KUKA KRL program: tool01_chk.src, tool01_chk.dat

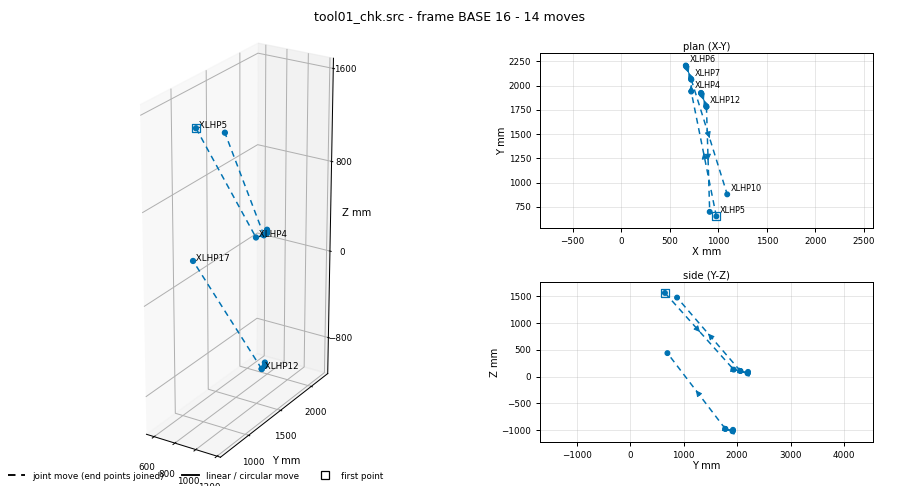
[picture p0: tool path of tool01_chk.src in frame BASE 16, 14 of 17 moves have a stored position in this frame; points joined in program order, loops and branches not executed]
--- tool01_chk.src ---
&ACCESS RVP
&REL 64
&COMMENT Werkzeugpruefprogramm
&PARAM TEMPLATE = C:\KRC\ROBOTER\TEMPLATE\VG_HP
&PARAM EDITMASK = *
DEF TOOL01_chk( )
;FOLD INI
;FOLD BASISTECH INI
    GLOBAL INTERRUPT DECL 3 WHEN $STOPMESS==TRUE DO IR_STOPM ( )
    INTERRUPT ON 3
    BAS (#INITMOV,0 )
;ENDFOLD (BASISTECH INI)
;FOLD SPOTTECH INI
    USERSPOT(#INIT)
;ENDFOLD (SPOTTECH INI)
;FOLD GRIPPERTECH INI
    USER_GRP(0,DUMMY,DUMMY,GDEFAULT)
;ENDFOLD (GRIPPERTECH INI)
;FOLD USER INI
;Make your modifications here
;FOLD COLLISION_V_3.01 INI ;%{E}
    IF (COLLISION_DATA[1].I_NR>0) THEN
    GLOBAL INTERRUPT DECL 21 WHEN $IN[COLLISION_DATA[1].I_NR]==FALSE DO COLLSTOP (1,0 )
    ENDIF
    IF (COLLISION_DATA[2].I_NR>0) THEN
    GLOBAL INTERRUPT DECL 22 WHEN $IN[COLLISION_DATA[2].I_NR]==FALSE DO COLLSTOP (2,0 )
    ENDIF
    IF (COLLISION_DATA[3].I_NR>0) THEN
    GLOBAL INTERRUPT DECL 23 WHEN $IN[COLLISION_DATA[3].I_NR]==FALSE DO COLLSTOP (3,0 )
    ENDIF
    IF (COLLISION_DATA[4].I_NR>0) THEN
    GLOBAL INTERRUPT DECL 24 WHEN $IN[COLLISION_DATA[4].I_NR]==FALSE DO COLLSTOP (4,0 )
    ENDIF
;ENDFOLD (Collision)
;ENDFOLD (USER INI)
;ENDFOLD (INI)
;FOLD ; Anlagenbezeichn:               Stations-Nr:;%{PE}%R 5.2.7,%MKUKATPBASIS,%CCOMMENT,%VNORMAL,%P 2:Anlagenbezeichn:               Stations-Nr:
;ENDFOLD
;FOLD ; Stand / Version:;%{PE}%R 5.2.7,%MKUKATPBASIS,%CCOMMENT,%VNORMAL,%P 2:Stand / Version:
;ENDFOLD
;FOLD ; Name Bearbeiter:;%{PE}%R 5.2.7,%MKUKATPBASIS,%CCOMMENT,%VNORMAL,%P 2:Name Bearbeiter:
;ENDFOLD
;Sicherheitsfrage (nur im Musterprogramm, nach teachen entfernen)
wait for false
;FOLD ; ***************************************;%{PE}%R 2.4.6,%MKUKATPBASIS,%CCOMMENT,%VNORMAL,%P 2:***************************************
;ENDFOLD
;FOLD ; A C H T U N G  ! ! !   Nur in T1 fahren;%{PE}%R 2.4.6,%MKUKATPBASIS,%CCOMMENT,%VNORMAL,%P 2:A C H T U N G  ! ! !   Nur in T1 fahren
;ENDFOLD
;FOLD ; ***************************************;%{PE}%R 2.4.6,%MKUKATPBASIS,%CCOMMENT,%VNORMAL,%P 2:***************************************
;ENDFOLD
WAIT FOR $T1
;Wenn notwendig vorher das Werkzeug im Bahnhof ablegen
;Roboterpruefprogramm
rob_ok ( )
;Wenn notwendig zu pruefendes Werkzeug ankoppeln
;FOLD PTP HOME  Vel= 100 % DEFAULT;%{PE}%R 3.2.43,%MKUKATPBASIS,%CMOVE,%VPTP,%P 1:PTP, 2:HOME, 3:, 5:100, 7:DEFAULT
$BWDSTART = FALSE
PDAT_ACT=PDEFAULT
BAS(#PTP_DAT)
FDAT_ACT=FHOME
BAS(#FRAMES)
BAS(#VEL_PTP,100)
$H_POS=XHOME
PTP XHOME
;ENDFOLD
;FOLD PTP LHP5  Vel= 100 % PDAT Tool[16] Base[16];%{PE}%R 3.2.43,%MKUKATPBASIS,%CMOVE,%VPTP,%P 1:PTP, 2:LHP5, 3:, 5:100, 7:PDAT
    $BWDSTART = FALSE
    PDAT_ACT=PPDAT
    BAS(#PTP_DAT)
    FDAT_ACT=FLHP5
    BAS(#FRAMES)
    BAS(#VEL_PTP,100)
    PTP XLHP5
;ENDFOLD
;FOLD PTP LHP4  Vel= 100 % PDAT Tool[16] Base[16];%{PE}%R 3.2.43,%MKUKATPBASIS,%CMOVE,%VPTP,%P 1:PTP, 2:LHP4, 3:, 5:100, 7:PDAT
    $BWDSTART = FALSE
    PDAT_ACT=PPDAT
    BAS(#PTP_DAT)
    FDAT_ACT=FLHP4
    BAS(#FRAMES)
    BAS(#VEL_PTP,100)
    PTP XLHP4
;ENDFOLD
;FOLD PTP LHP7  Vel= 100 % PDAT Tool[16] Base[16];%{PE}%R 3.2.43,%MKUKATPBASIS,%CMOVE,%VPTP,%P 1:PTP, 2:LHP7, 3:, 5:100, 7:PDAT
    $BWDSTART = FALSE
    PDAT_ACT=PPDAT
    BAS(#PTP_DAT)
    FDAT_ACT=FLHP7
    BAS(#FRAMES)
    BAS(#VEL_PTP,100)
    PTP XLHP7
;ENDFOLD
;FOLD PTP LHP6  Vel= 100 % PDAT Tool[16] Base[16];%{PE}%R 3.2.43,%MKUKATPBASIS,%CMOVE,%VPTP,%P 1:PTP, 2:LHP6, 3:, 5:100, 7:PDAT
    $BWDSTART = FALSE
    PDAT_ACT=PPDAT
    BAS(#PTP_DAT)
    FDAT_ACT=FLHP6
    BAS(#FRAMES)
    BAS(#VEL_PTP,100)
    PTP XLHP6
;ENDFOLD
;FOLD ; 1.Kontrollposition mit Tool 16;%{PE}%R 5.2.17,%MKUKATPBASIS,%CCOMMENT,%VNORMAL,%P 2:1.Kontrollposition mit Tool 16
;ENDFOLD
;FOLD ; Pruefspitze - Werkzeugspitze bzw. Greiferreferenzpunkt;%{PE}%R 2.4.6,%MKUKATPBASIS,%CCOMMENT,%VNORMAL,%P 2:Pruefspitze - Werkzeugspitze bzw. Greiferreferenzpunkt
;ENDFOLD
;FOLD ; Spitze unten;%{PE}%R 2.4.6,%MKUKATPBASIS,%CCOMMENT,%VNORMAL,%P 2:Spitze unten
;ENDFOLD
;FOLD LIN Kontroll1  Vel= 1 m/s CPDAT Tool[16] Base[16];%{PE}%R 3.2.43,%MKUKATPBASIS,%CMOVE,%VLIN,%P 1:LIN, 2:Kontroll1, 3:, 5:1, 7:CPDAT
    $BWDSTART = FALSE
    LDAT_ACT=LCPDAT
    BAS(#CP_DAT)
    FDAT_ACT=FKontroll1
    BAS(#FRAMES)
    BAS(#VEL_CP,1)
    LIN XKontroll1
;ENDFOLD
WAIT FOR  $IN[1026]==TRUE ; Kontrollposition Werkzeug mit Tool16 (Nullwerkzeug)
;PTP LHP freifahren
;FOLD LIN LHP8  Vel= 2 m/s CPDAT Tool[16] Base[16];%{PE}%R 3.2.43,%MKUKATPBASIS,%CMOVE,%VLIN,%P 1:LIN, 2:LHP8, 3:, 5:2, 7:CPDAT
    $BWDSTART = FALSE
    LDAT_ACT=LCPDAT
    BAS(#CP_DAT)
    FDAT_ACT=FLHP8
    BAS(#FRAMES)
    BAS(#VEL_CP,2)
    LIN XLHP8
;ENDFOLD
;FOLD PTP LHP9  Vel= 100 % PDAT Tool[16] Base[16];%{PE}%R 3.2.43,%MKUKATPBASIS,%CMOVE,%VPTP,%P 1:PTP, 2:LHP9, 3:, 5:100, 7:PDAT
    $BWDSTART = FALSE
    PDAT_ACT=PPDAT
    BAS(#PTP_DAT)
    FDAT_ACT=FLHP9
    BAS(#FRAMES)
    BAS(#VEL_PTP,100)
    PTP XLHP9
;ENDFOLD
;FOLD PTP LHP10  Vel= 100 % PDAT Tool[16] Base[16];%{PE}%R 3.2.43,%MKUKATPBASIS,%CMOVE,%VPTP,%P 1:PTP, 2:LHP10, 3:, 5:100, 7:PDAT
    $BWDSTART = FALSE
    PDAT_ACT=PPDAT
    BAS(#PTP_DAT)
    FDAT_ACT=FLHP10
    BAS(#FRAMES)
    BAS(#VEL_PTP,100)
    PTP XLHP10
;ENDFOLD
;Wichtig: auf Home zurueck fahren und auf aktuelles TOOL umschalten
;FOLD PTP HOME  Vel= 100 % PDAT;%{PE}%R 3.2.43,%MKUKATPBASIS,%CMOVE,%VPTP,%P 1:PTP, 2:HOME, 3:, 5:100, 7:PDAT
    $BWDSTART = FALSE
    PDAT_ACT=PPDAT
    BAS(#PTP_DAT)
    FDAT_ACT=FHOME
    BAS(#FRAMES)
    BAS(#VEL_PTP,100)
    $H_POS=XHOME
    PTP XHOME
;ENDFOLD
;FOLD PTP LHP12  Vel= 100 % PDAT Tool[1] Base[16];%{PE}%R 3.2.43,%MKUKATPBASIS,%CMOVE,%VPTP,%P 1:PTP, 2:LHP12, 3:, 5:100, 7:PDAT
    $BWDSTART = FALSE
    PDAT_ACT=PPDAT
    BAS(#PTP_DAT)
    FDAT_ACT=FLHP12
    BAS(#FRAMES)
    BAS(#VEL_PTP,100)
    PTP XLHP12
;ENDFOLD
;FOLD PTP LHP13  Vel= 100 % PDAT Tool[1] Base[16];%{PE}%R 3.2.43,%MKUKATPBASIS,%CMOVE,%VPTP,%P 1:PTP, 2:LHP13, 3:, 5:100, 7:PDAT
    $BWDSTART = FALSE
    PDAT_ACT=PPDAT
    BAS(#PTP_DAT)
    FDAT_ACT=FLHP13
    BAS(#FRAMES)
    BAS(#VEL_PTP,100)
    PTP XLHP13
;ENDFOLD
;FOLD ; 2.Kontrollposition mit Tool aktuell;%{PE}%R 5.2.17,%MKUKATPBASIS,%CCOMMENT,%VNORMAL,%P 2:2.Kontrollposition mit Tool aktuell
;ENDFOLD
;FOLD ; Pruefspitze - Werkzeugspitze bzw. Greiferreferenzpunkt;%{PE}%R 2.4.6,%MKUKATPBASIS,%CCOMMENT,%VNORMAL,%P 2:Pruefspitze - Werkzeugspitze bzw. Greiferreferenzpunkt
;ENDFOLD
;FOLD ; Spitze unten;%{PE}%R 2.4.6,%MKUKATPBASIS,%CCOMMENT,%VNORMAL,%P 2:Spitze unten
;ENDFOLD
;PTP KONTROLL2 teachen mit dem zugehoerigen Tool
;FOLD LIN Kontroll2  Vel= 1 m/s CPDAT Tool[1] Base[16];%{PE}%R 3.2.43,%MKUKATPBASIS,%CMOVE,%VLIN,%P 1:LIN, 2:Kontroll2, 3:, 5:1, 7:CPDAT
    $BWDSTART = FALSE
    LDAT_ACT=LCPDAT
    BAS(#CP_DAT)
    FDAT_ACT=FKontroll2
    BAS(#FRAMES)
    BAS(#VEL_CP,1)
    LIN XKontroll2
;ENDFOLD
WAIT FOR  $IN[1026]==TRUE ; Kontrollposition Werkzeug mit zugehoerigem Tool
;PTP LHP zur Ausgangsstellung
;FOLD LIN LHP15  Vel= 1 m/s CPDAT Tool[1] Base[16];%{PE}%R 3.2.43,%MKUKATPBASIS,%CMOVE,%VLIN,%P 1:LIN, 2:LHP15, 3:, 5:1, 7:CPDAT
    $BWDSTART = FALSE
    LDAT_ACT=LCPDAT
    BAS(#CP_DAT)
    FDAT_ACT=FLHP15
    BAS(#FRAMES)
    BAS(#VEL_CP,1)
    LIN XLHP15
;ENDFOLD
;FOLD PTP LHP16  Vel= 100 % PDAT Tool[1] Base[16];%{PE}%R 3.2.43,%MKUKATPBASIS,%CMOVE,%VPTP,%P 1:PTP, 2:LHP16, 3:, 5:100, 7:PDAT
    $BWDSTART = FALSE
    PDAT_ACT=PPDAT
    BAS(#PTP_DAT)
    FDAT_ACT=FLHP16
    BAS(#FRAMES)
    BAS(#VEL_PTP,100)
    PTP XLHP16
;ENDFOLD
;FOLD PTP LHP17  Vel= 100 % PDAT Tool[1] Base[16];%{PE}%R 3.2.43,%MKUKATPBASIS,%CMOVE,%VPTP,%P 1:PTP, 2:LHP17, 3:, 5:100, 7:PDAT
    $BWDSTART = FALSE
    PDAT_ACT=PPDAT
    BAS(#PTP_DAT)
    FDAT_ACT=FLHP17
    BAS(#FRAMES)
    BAS(#VEL_PTP,100)
    PTP XLHP17
;ENDFOLD
;FOLD PTP HOME  Vel= 100 % DEFAULT;%{PE}%R 3.2.43,%MKUKATPBASIS,%CMOVE,%VPTP,%P 1:PTP, 2:HOME, 3:, 5:100, 7:DEFAULT
    $BWDSTART = FALSE
    PDAT_ACT=PDEFAULT
    BAS(#PTP_DAT)
    FDAT_ACT=FHOME
    BAS(#FRAMES)
    BAS(#VEL_PTP,100)
    $H_POS=XHOME
    PTP XHOME
;ENDFOLD
;Wenn notwendig das ursprüngliche Werkzeug wieder ankoppeln
END

--- tool01_chk.dat ---
&ACCESS RVP
&REL 64
&COMMENT Werkzeugpruefprogramm
&PARAM TEMPLATE = C:\KRC\ROBOTER\TEMPLATE\VG_HP
&PARAM EDITMASK = *
DEFDAT  TOOL01_CHK
;FOLD EXTERNAL DECLARATIONS;%{PE}%V3.2.0,%MKUKATPBASIS,%CEXT,%VCOMMON,%P
;ENDFOLD

DECL BASIS_SUGG_T LAST_BASIS={POINT1[] "P0                      ",POINT2[] "P0                      ",CP_PARAMS[] "CPDAT0                  ",PTP_PARAMS[] "PDAT0                  ",CONT[] "                        ",CP_VEL[] "2                       ",PTP_VEL[] "100                     "}
DECL E6POS XLHP1={x 980.162,y 652.3817,z 1564.854,a 159.7475,b -4.016941,c 179.1242,s 18,t 43,e1 -100.6665,e2 0.0,e3 0.0,e4 0.0,e5 0.0,e6 0.0}
DECL E6POS XKONTROLL1={x 665.4379,y 2205.945,z 89.04919,a -69.02276,b -16.31656,c -177.4203,s 18,t 3,e1 -100.6661,e2 0.0,e3 0.0,e4 0.0,e5 0.0,e6 0.0}
DECL E6POS XLHP4={x 721.3241,y 1937.913,z 131.173,a -69.07279,b -16.22725,c -174.2469,s 18,t 3,e1 -100.6665,e2 0.0,e3 0.0,e4 0.0,e5 0.0,e6 0.0}
DECL E6POS XLHP5={x 980.1787,y 652.3956,z 1564.878,a 159.749,b -4.016594,c 179.1235,s 18,t 43,e1 -100.6665,e2 0.0,e3 0.0,e4 0.0,e5 0.0,e6 0.0}
DECL E6POS XKONTROLL2={x 821.7288,y 1924.512,z -993.7808,a 111.0075,b 16.30128,c -2.863059,s 18,t 3,e1 -100.6665,e2 0.0,e3 0.0,e4 0.0,e5 0.0,e6 0.0}
DECL E6POS XLHP6={x 669.3153,y 2199.305,z 63.11586,a -69.03085,b -16.31788,c -177.4184,s 18,t 3,e1 -100.6665,e2 0.0,e3 0.0,e4 0.0,e5 0.0,e6 0.0}
DECL E6POS XLHP7={x 721.9332,y 2061.901,z 106.2138,a -69.02566,b -16.3192,c -177.4167,s 18,t 3,e1 -100.6665,e2 0.0,e3 0.0,e4 0.0,e5 0.0,e6 0.0}
DECL E6POS XLHP8={x 669.3173,y 2199.294,z 63.11121,a -69.03092,b -16.31823,c -177.4184,s 18,t 3,e1 -100.6665,e2 0.0,e3 0.0,e4 0.0,e5 0.0,e6 0.0}
DECL E6POS XLHP9={x 721.9332,y 2061.901,z 106.2138,a -69.02566,b -16.3192,c -177.4167,s 18,t 3,e1 -100.6665,e2 0.0,e3 0.0,e4 0.0,e5 0.0,e6 0.0}
DECL E6POS XLHP10={x 1092.313,y 878.8538,z 1478.174,a 177.4667,b -3.04429,c -178.5137,s 18,t 43,e1 -100.6665,e2 0.0,e3 0.0,e4 0.0,e5 0.0,e6 0.0}
DECL E6POS XLHP12={x 878.2603,y 1780.715,z -976.2581,a 111.0027,b 16.29478,c -2.869996,s 18,t 3,e1 -100.6665,e2 0.0,e3 0.0,e4 0.0,e5 0.0,e6 0.0}
DECL E6POS XLHP13={x 825.5921,y 1917.879,z -1019.667,a 111.0074,b 16.30032,c -2.863573,s 18,t 3,e1 -100.6665,e2 0.0,e3 0.0,e4 0.0,e5 0.0,e6 0.0}
DECL E6POS XLHP15={x 825.5995,y 1917.881,z -1019.669,a 111.007,b 16.29994,c -2.863638,s 18,t 3,e1 -100.6665,e2 0.0,e3 0.0,e4 0.0,e5 0.0,e6 0.0}
DECL E6POS XLHP16={x 878.2797,y 1780.88,z -976.2927,a 111.0091,b 16.29242,c -2.869744,s 18,t 3,e1 -100.6665,e2 0.0,e3 0.0,e4 0.0,e5 0.0,e6 0.0}
DECL E6POS XLHP17={x 911.847,y 698.7325,z 439.7753,a -20.25009,b 3.988059,c 0.4698318,s 18,t 43,e1 -100.6665,e2 0.0,e3 0.0,e4 0.0,e5 0.0,e6 0.0}
DECL FDAT FLHP1={TOOL_NO 16,BASE_NO 16,IPO_FRAME #BASE}
DECL FDAT FKONTROLL1={TOOL_NO 16,BASE_NO 16,IPO_FRAME #BASE}
DECL FDAT FLHP4={TOOL_NO 16,BASE_NO 16,IPO_FRAME #BASE}
DECL FDAT FLHP5={TOOL_NO 16,BASE_NO 16,IPO_FRAME #BASE}
DECL FDAT FKontroll2={TOOL_NO 1,BASE_NO 16,IPO_FRAME #BASE}
DECL FDAT FLHP6={TOOL_NO 16,BASE_NO 16,IPO_FRAME #BASE}
DECL FDAT FLHP7={TOOL_NO 16,BASE_NO 16,IPO_FRAME #BASE}
DECL FDAT FLHP8={TOOL_NO 16,BASE_NO 16,IPO_FRAME #BASE}
DECL FDAT FLHP9={TOOL_NO 16,BASE_NO 16,IPO_FRAME #BASE}
DECL FDAT FLHP10={TOOL_NO 16,BASE_NO 16,IPO_FRAME #BASE}
DECL FDAT FLHP12={TOOL_NO 1,BASE_NO 16,IPO_FRAME #BASE}
DECL FDAT FLHP13={TOOL_NO 1,BASE_NO 16,IPO_FRAME #BASE}
DECL FDAT FLHP15={TOOL_NO 1,BASE_NO 16,IPO_FRAME #BASE}
DECL FDAT FLHP16={TOOL_NO 1,BASE_NO 16,IPO_FRAME #BASE}
DECL FDAT FLHP17={TOOL_NO 1,BASE_NO 16,IPO_FRAME #BASE}
DECL FDAT FHOME={TOOL_NO 1,BASE_NO 0,IPO_FRAME #BASE}
DECL PDAT PPDAT={VEL 100.0,ACC 100.0,APO_DIST 100.0}
DECL LDAT LCPDAT={VEL 2.0,ACC 100.0,APO_DIST 100.0,APO_FAC 50.0}
ENDDAT
